Staubli VAL3: CmdDeal.pgx

program CmdDeal()
  local num ln_i
  local num ln_total
  local string strX
  local string strY
  local num nPosX
  local num nPosY
  local bool bOk
  local num nPosZ
  local string strZ
  local num local1
  local string strAct
  local num nAct
  local bool bTemp
  local joint jTemp1
begin
  while true
    //deal the command from another robot
    if nReadPt!=nWritePt
      strCmd=mid(CmdBuffer[nReadPt],6,1)

      if strCmd=="RBNEXT"
        TcpStrRec:nCtrl=0
      endIf
      if strCmd=="RBHOME"
        bRb2Home=true
        bRb2Ready=false
      endIf
      if strCmd=="RBREDY"
        popUpMsg("okl")
        bRb2Ready=true
        bRb2Home=false
      endIf
      if strCmd=="RBSTOP"
        bRb2Ready=false
        bRb2Home=false
        bRb2Stop=true
        bRb2Start=false
        bSychronOn=false
      endIf
      if strCmd=="RBSTAT"
        bRb2Home=false
        bRb2Stop=false
        bRb2Start=true
        bSychronOn=true
      endIf
      if strCmd=="RBINIT"
        bRb2InitOk=true
      endIf
      if strCmd=="RBAXI8"
        bRb2AXI8=true
      endIf
      CmdBuffer[nReadPt]=""
      CmdTotal=CmdTotal-1
      nReadPt=nReadPt+1
      if nReadPt>=20
        nReadPt=0
      endIf
    endIf
    delay(0)
  endWhile
end
